TYPE E_TCPIP_State_1 :
(
	E_TCPIP_IDLE,
	E_TCPIP_CONNECT,
	E_TCPIP_SEND,
	E_TCPIP_RECEIVE,
	E_TCPIP_DISCONNECT,
	E_TCPIP_CLOSEALL,
	E_TCPIP_DONE
);
END_TYPE

(* stored: Version 1.1.0.1
   DUT E_TCPIP_State_1: Id {213315cb-5cc3-4380-87cb-c673a32a2b69} *)
